// TIA Portal V19 export
TYPE "PII - CSS 01411.2-xx"
   STRUCT
      "Process Data Inputs - Temperature" : Int;
      "Process Data Inputs - Temperature Alarm High" : Bool;
      "Process Data Inputs - Temperature Range High" : Bool;
      "Process Data Inputs - Temperature Range Low" : Bool;
      "Process Data Inputs - Temperature Alarm Low" : Bool;
      "Reserved Bit" : Bool;
      "Reserved Bit_1" : Bool;
      "Reserved Bit_2" : Bool;
      "Reserved Bit_3" : Bool;
      "Process Data Inputs - Humidity" : Int;
      "Process Data Inputs - Humidity Alarm High" : Bool;
      "Process Data Inputs - Humidity Range High" : Bool;
      "Process Data Inputs - Humidity Range Low" : Bool;
      "Process Data Inputs - Humidity Alarm Low" : Bool;
      "Reserved Bit_4" : Bool;
      "Reserved Bit_5" : Bool;
      "Reserved Bit_6" : Bool;
      "Reserved Bit_7" : Bool;
      "Reserved Byte" : Bool;
      "Reserved Byte_1" : Bool;
      "Reserved Byte_2" : Bool;
      "Reserved Byte_3" : Bool;
      "Reserved Byte_4" : Bool;
      "Reserved Byte_5" : Bool;
      "Reserved Byte_6" : Bool;
      "Reserved Byte_7" : Bool;
      "Reserved Byte_8" : Bool;
      "Reserved Byte_9" : Bool;
      "Reserved Byte_10" : Bool;
      "Reserved Byte_11" : Bool;
      "Reserved Byte_12" : Bool;
      "Reserved Byte_13" : Bool;
      "Reserved Byte_14" : Bool;
      "Reserved Byte_15" : Bool;
      "Reserved Byte_16" : Bool;
      "Reserved Byte_17" : Bool;
      "Reserved Byte_18" : Bool;
      "Reserved Byte_19" : Bool;
      "Reserved Byte_20" : Bool;
      "Reserved Byte_21" : Bool;
      "Reserved Byte_22" : Bool;
      "Reserved Byte_23" : Bool;
      "Reserved Byte_24" : Bool;
      "Reserved Byte_25" : Bool;
      "Port qualifier" : Byte;
   END_STRUCT;
END_TYPE
